(* IEC 61131-3 sources: 3D-Asset-Platform-V2/openplc/cobot-6dof-smart-demo, 5 files *)

(* ---- cobot_6dof_iot_condition_monitoring.st ---- *)
VAR
  Command AT %QW90 : UINT := 0;
  Status AT %QW91 : UINT := 0;
  ActiveStep AT %QW92 : UINT := 0;
  ElapsedMsOut AT %QW93 : UINT := 0;
  AlarmCode AT %QW94 : UINT := 0;
  ConditionState AT %QW95 : UINT := 3;
  SpeedPermille AT %QW96 : UINT := 0;
  J1Raw AT %QW100 : INT := 0;
  J2Raw AT %QW101 : INT := -6109;
  J3Raw AT %QW102 : INT := 13090;
  J4Raw AT %QW103 : INT := 8727;
  J5Raw AT %QW104 : INT := 0;
  J6Raw AT %QW105 : INT := 0;
  TemperatureCx100 AT %QW120 : INT := 0;
  HumidityRHx100 AT %QW121 : UINT := 0;
  GyroDpsx100 AT %QW122 : UINT := 0;
  SensorAgeMs AT %QW123 : UINT := 65535;
  SensorValid AT %QW124 : UINT := 0;
  SensorSequence AT %QW125 : UINT := 0;
  SensorQualityBits AT %QW126 : UINT := 0;
  SensorPolicy AT %QW127 : UINT := 1;
  CycleTimer : TON;
  MotionIdleTimer : TON;
  TimerEnabled : BOOL := FALSE;
  ResetTimer : BOOL := TRUE;
  ElapsedMs : DINT := 0;
  SegmentStartMs : DINT := 0;
  SegmentDurationMs : DINT := 1;
  P : REAL := 0.0;
  MotionScale : REAL := 1.0;
  TemperatureC : REAL := 0.0;
  HumidityRH : REAL := 0.0;
  GyroDps : REAL := 0.0;
  J1Deg : REAL := 0.0;
  J2Deg : REAL := -35.0;
  J3Deg : REAL := 75.0;
  J4Deg : REAL := 50.0;
  J5Deg : REAL := 0.0;
  J6Deg : REAL := 0.0;
  TargetJ1 : REAL := 0.0;
  TargetJ2 : REAL := -35.0;
  TargetJ3 : REAL := 75.0;
  TargetJ4 : REAL := 50.0;
  TargetJ5 : REAL := 0.0;
  TargetJ6 : REAL := 0.0;
  MotionPresent : BOOL := FALSE;
  DegToRadScaled : REAL := 174.5329;
END_VAR

TemperatureC := INT_TO_REAL(TemperatureCx100) / 100.0;
HumidityRH := UINT_TO_REAL(HumidityRHx100) / 100.0;
GyroDps := UINT_TO_REAL(GyroDpsx100) / 100.0;
MotionPresent := GyroDps >= 3.0;
MotionIdleTimer(IN := (SensorPolicy = 1) AND (NOT MotionPresent), PT := T#2s);

ConditionState := 0;
AlarmCode := 0;
MotionScale := 1.0;
SpeedPermille := 1000;

IF (SensorValid = 0) OR ((SensorQualityBits AND 1) = 0) OR (SensorAgeMs > 2500) THEN
  ConditionState := 3;
  AlarmCode := 4;
  MotionScale := 0.0;
  SpeedPermille := 0;
ELSIF (SensorPolicy = 1) AND ((SensorQualityBits AND 16) = 0) THEN
  ConditionState := 3;
  AlarmCode := 6;
  MotionScale := 0.0;
  SpeedPermille := 0;
ELSIF (SensorPolicy = 1) AND MotionIdleTimer.Q THEN
  ConditionState := 2;
  AlarmCode := 5;
  MotionScale := 0.0;
  SpeedPermille := 0;
ELSIF (TemperatureC >= 55.0) OR (HumidityRH >= 85.0) OR (GyroDps >= 220.0) THEN
  ConditionState := 2;
  MotionScale := 0.0;
  SpeedPermille := 0;
  IF TemperatureC >= 55.0 THEN
    AlarmCode := 1;
  ELSIF HumidityRH >= 85.0 THEN
    AlarmCode := 2;
  ELSE
    AlarmCode := 3;
  END_IF;
ELSIF (TemperatureC >= 45.0) OR (HumidityRH >= 75.0) OR (GyroDps >= 120.0) THEN
  ConditionState := 1;
  MotionScale := 0.55;
  SpeedPermille := 550;
END_IF;

IF Command = 2 THEN
  TimerEnabled := FALSE;
  ResetTimer := TRUE;
  Status := 2;
  ActiveStep := 0;
  ElapsedMsOut := 0;
  J1Deg := 0.0;
  J2Deg := -35.0;
  J3Deg := 75.0;
  J4Deg := 50.0;
  J5Deg := 0.0;
  J6Deg := 0.0;
ELSIF Command = 0 THEN
  TimerEnabled := FALSE;
  ResetTimer := TRUE;
  Status := 0;
  ActiveStep := 0;
  J1Deg := INT_TO_REAL(J1Raw) / DegToRadScaled;
  J2Deg := INT_TO_REAL(J2Raw) / DegToRadScaled;
  J3Deg := INT_TO_REAL(J3Raw) / DegToRadScaled;
  J4Deg := INT_TO_REAL(J4Raw) / DegToRadScaled;
  J5Deg := INT_TO_REAL(J5Raw) / DegToRadScaled;
  J6Deg := INT_TO_REAL(J6Raw) / DegToRadScaled;
ELSIF ConditionState >= 2 THEN
  TimerEnabled := FALSE;
  ResetTimer := TRUE;
  Status := 3;
  ActiveStep := 0;
ELSE
  Status := 1;
  IF ResetTimer THEN
    TimerEnabled := FALSE;
    ResetTimer := FALSE;
  ELSE
    TimerEnabled := TRUE;
  END_IF;

  CycleTimer(IN := TimerEnabled, PT := T#12s);
  ElapsedMs := TIME_TO_DINT(CycleTimer.ET);
  IF ElapsedMs > 12000 THEN ElapsedMs := 12000; END_IF;
  ElapsedMsOut := DINT_TO_UINT(ElapsedMs);

  IF ElapsedMs < 3000 THEN
    ActiveStep := 1; SegmentStartMs := 0; SegmentDurationMs := 3000;
    TargetJ1 := -90.0; TargetJ2 := -10.0; TargetJ3 := 105.0;
    TargetJ4 := 10.0; TargetJ5 := -45.0; TargetJ6 := -90.0;
  ELSIF ElapsedMs < 6000 THEN
    ActiveStep := 2; SegmentStartMs := 3000; SegmentDurationMs := 3000;
    TargetJ1 := 90.0; TargetJ2 := 40.0; TargetJ3 := 125.0;
    TargetJ4 := -70.0; TargetJ5 := 60.0; TargetJ6 := 120.0;
  ELSIF ElapsedMs < 9000 THEN
    ActiveStep := 3; SegmentStartMs := 6000; SegmentDurationMs := 3000;
    TargetJ1 := -55.0; TargetJ2 := -75.0; TargetJ3 := 45.0;
    TargetJ4 := 120.0; TargetJ5 := -80.0; TargetJ6 := -140.0;
  ELSE
    ActiveStep := 4; SegmentStartMs := 9000; SegmentDurationMs := 3000;
    TargetJ1 := 0.0; TargetJ2 := -35.0; TargetJ3 := 75.0;
    TargetJ4 := 50.0; TargetJ5 := 0.0; TargetJ6 := 0.0;
  END_IF;

  P := DINT_TO_REAL(ElapsedMs - SegmentStartMs) / DINT_TO_REAL(SegmentDurationMs);
  IF P < 0.0 THEN P := 0.0; END_IF;
  IF P > 1.0 THEN P := 1.0; END_IF;
  P := P * P * (3.0 - (2.0 * P));

  J1Deg := J1Deg + (((0.0 + ((TargetJ1 - 0.0) * MotionScale)) - J1Deg) * P);
  J2Deg := J2Deg + (((-35.0 + ((TargetJ2 - (-35.0)) * MotionScale)) - J2Deg) * P);
  J3Deg := J3Deg + (((75.0 + ((TargetJ3 - 75.0) * MotionScale)) - J3Deg) * P);
  J4Deg := J4Deg + (((50.0 + ((TargetJ4 - 50.0) * MotionScale)) - J4Deg) * P);
  J5Deg := J5Deg + (((0.0 + ((TargetJ5 - 0.0) * MotionScale)) - J5Deg) * P);
  J6Deg := J6Deg + (((0.0 + ((TargetJ6 - 0.0) * MotionScale)) - J6Deg) * P);

  IF CycleTimer.Q THEN ResetTimer := TRUE; END_IF;
END_IF;

J1Raw := REAL_TO_INT(J1Deg * DegToRadScaled);
J2Raw := REAL_TO_INT(J2Deg * DegToRadScaled);
J3Raw := REAL_TO_INT(J3Deg * DegToRadScaled);
J4Raw := REAL_TO_INT(J4Deg * DegToRadScaled);
J5Raw := REAL_TO_INT(J5Deg * DegToRadScaled);
J6Raw := REAL_TO_INT(J6Deg * DegToRadScaled);

(* ---- cobot_6dof_smart_demo.st ---- *)
VAR
  Command AT %QW90 : UINT := 1;
  Status AT %QW91 : UINT := 1;
  ActiveStep AT %QW92 : UINT := 0;
  ElapsedMsOut AT %QW93 : UINT := 0;
  J1Raw AT %QW100 : INT := 0;
  J2Raw AT %QW101 : INT := -6109;
  J3Raw AT %QW102 : INT := 13090;
  J4Raw AT %QW103 : INT := 8727;
  J5Raw AT %QW104 : INT := 0;
  J6Raw AT %QW105 : INT := 0;
  CycleTimer : TON;
  TimerEnabled : BOOL := TRUE;
  ResetTimer : BOOL := FALSE;
  ElapsedMs : DINT := 0;
  SegmentStartMs : DINT := 0;
  SegmentDurationMs : DINT := 1;
  P : REAL := 0.0;
  J1Deg : REAL := 0.0;
  J2Deg : REAL := -35.0;
  J3Deg : REAL := 75.0;
  J4Deg : REAL := 50.0;
  J5Deg : REAL := 0.0;
  J6Deg : REAL := 0.0;
  DegToRadScaled : REAL := 174.5329;
END_VAR

IF Command = 2 THEN
  TimerEnabled := FALSE; Status := 2; ActiveStep := 0; ElapsedMsOut := 0;
  J1Deg := 0.0; J2Deg := -35.0; J3Deg := 75.0;
  J4Deg := 50.0; J5Deg := 0.0; J6Deg := 0.0;
ELSIF Command = 0 THEN
  TimerEnabled := FALSE; Status := 0; ActiveStep := 0;
  J1Deg := INT_TO_REAL(J1Raw) / DegToRadScaled;
  J2Deg := INT_TO_REAL(J2Raw) / DegToRadScaled;
  J3Deg := INT_TO_REAL(J3Raw) / DegToRadScaled;
  J4Deg := INT_TO_REAL(J4Raw) / DegToRadScaled;
  J5Deg := INT_TO_REAL(J5Raw) / DegToRadScaled;
  J6Deg := INT_TO_REAL(J6Raw) / DegToRadScaled;
ELSE
  Status := 1;
  IF ResetTimer THEN
    TimerEnabled := FALSE; ResetTimer := FALSE;
  ELSE
    TimerEnabled := TRUE;
  END_IF;

  CycleTimer(IN := TimerEnabled, PT := T#10s);
  ElapsedMs := TIME_TO_DINT(CycleTimer.ET);
  IF ElapsedMs > 10000 THEN ElapsedMs := 10000; END_IF;
  ElapsedMsOut := DINT_TO_UINT(ElapsedMs);

  IF ElapsedMs < 1400 THEN
    ActiveStep := 1; SegmentStartMs := 0; SegmentDurationMs := 1400;
  ELSIF ElapsedMs < 2400 THEN
    ActiveStep := 2; SegmentStartMs := 1400; SegmentDurationMs := 1000;
  ELSIF ElapsedMs < 3200 THEN
    ActiveStep := 3; SegmentStartMs := 2400; SegmentDurationMs := 800;
  ELSIF ElapsedMs < 5600 THEN
    ActiveStep := 4; SegmentStartMs := 3200; SegmentDurationMs := 2400;
  ELSIF ElapsedMs < 7600 THEN
    ActiveStep := 5; SegmentStartMs := 5600; SegmentDurationMs := 2000;
  ELSE
    ActiveStep := 6; SegmentStartMs := 7600; SegmentDurationMs := 2400;
  END_IF;

  IF SegmentDurationMs > 0 THEN
    P := DINT_TO_REAL(ElapsedMs - SegmentStartMs) / DINT_TO_REAL(SegmentDurationMs);
    IF P < 0.0 THEN P := 0.0; ELSIF P > 1.0 THEN P := 1.0; END_IF;
    P := P * P * (3.0 - (2.0 * P));
  ELSE
    P := 0.0;
  END_IF;

  IF ActiveStep = 1 THEN
    J1Deg := 0.0 + ((-55.0 - 0.0) * P);
    J2Deg := -35.0 + ((-10.0 - (-35.0)) * P);
    J3Deg := 75.0 + ((85.0 - 75.0) * P);
    J4Deg := 50.0 + ((25.0 - 50.0) * P);
    J5Deg := 0.0;
    J6Deg := 0.0;
  ELSIF ActiveStep = 2 THEN
    J1Deg := -55.0;
    J2Deg := -10.0 + ((15.0 - (-10.0)) * P);
    J3Deg := 85.0 + ((80.0 - 85.0) * P);
    J4Deg := 25.0 + ((-5.0 - 25.0) * P);
    J5Deg := 0.0;
    J6Deg := 0.0;
  ELSIF ActiveStep = 3 THEN
    J1Deg := -55.0;
    J2Deg := 15.0;
    J3Deg := 80.0;
    J4Deg := -5.0;
    J5Deg := 0.0;
    J6Deg := 0.0 + ((90.0 - 0.0) * P);
  ELSIF ActiveStep = 4 THEN
    J1Deg := -55.0 + ((50.0 - (-55.0)) * P);
    J2Deg := 15.0 + ((-10.0 - 15.0) * P);
    J3Deg := 80.0 + ((85.0 - 80.0) * P);
    J4Deg := -5.0 + ((25.0 - (-5.0)) * P);
    J5Deg := 0.0;
    J6Deg := 90.0;
  ELSIF ActiveStep = 5 THEN
    J1Deg := 50.0;
    J2Deg := -10.0 + ((15.0 - (-10.0)) * P);
    J3Deg := 85.0 + ((80.0 - 85.0) * P);
    J4Deg := 25.0 + ((-5.0 - 25.0) * P);
    J5Deg := 0.0 + ((30.0 - 0.0) * P);
    J6Deg := 90.0 + ((-90.0 - 90.0) * P);
  ELSE
    J1Deg := 50.0 + ((0.0 - 50.0) * P);
    J2Deg := 15.0 + ((-35.0 - 15.0) * P);
    J3Deg := 80.0 + ((75.0 - 80.0) * P);
    J4Deg := -5.0 + ((50.0 - (-5.0)) * P);
    J5Deg := 30.0 + ((0.0 - 30.0) * P);
    J6Deg := -90.0 + ((0.0 - (-90.0)) * P);
  END_IF;

  IF CycleTimer.Q THEN ResetTimer := TRUE; END_IF;
END_IF;

J1Raw := REAL_TO_INT(J1Deg * DegToRadScaled);
J2Raw := REAL_TO_INT(J2Deg * DegToRadScaled);
J3Raw := REAL_TO_INT(J3Deg * DegToRadScaled);
J4Raw := REAL_TO_INT(J4Deg * DegToRadScaled);
J5Raw := REAL_TO_INT(J5Deg * DegToRadScaled);
J6Raw := REAL_TO_INT(J6Deg * DegToRadScaled);

(* ---- cobot_6dof_smart_demo_amplified.st ---- *)
VAR
  Command AT %QW90 : UINT := 0;
  Status AT %QW91 : UINT := 0;
  ActiveStep AT %QW92 : UINT := 0;
  ElapsedMsOut AT %QW93 : UINT := 0;
  J1Raw AT %QW100 : INT := 0;
  J2Raw AT %QW101 : INT := -6109;
  J3Raw AT %QW102 : INT := 13090;
  J4Raw AT %QW103 : INT := 8727;
  J5Raw AT %QW104 : INT := 0;
  J6Raw AT %QW105 : INT := 0;
  CycleTimer : TON;
  TimerEnabled : BOOL := FALSE;
  ResetTimer : BOOL := FALSE;
  ElapsedMs : DINT := 0;
  SegmentStartMs : DINT := 0;
  SegmentDurationMs : DINT := 1;
  P : REAL := 0.0;
  J1Deg : REAL := 0.0;
  J2Deg : REAL := -35.0;
  J3Deg : REAL := 75.0;
  J4Deg : REAL := 50.0;
  J5Deg : REAL := 0.0;
  J6Deg : REAL := 0.0;
  DegToRadScaled : REAL := 174.5329;
END_VAR

IF Command = 2 THEN
  TimerEnabled := FALSE;
  ResetTimer := TRUE;
  Status := 2;
  ActiveStep := 0;
  ElapsedMsOut := 0;
  J1Deg := 0.0;
  J2Deg := -35.0;
  J3Deg := 75.0;
  J4Deg := 50.0;
  J5Deg := 0.0;
  J6Deg := 0.0;
ELSIF Command = 0 THEN
  TimerEnabled := FALSE;
  ResetTimer := TRUE;
  Status := 0;
  ActiveStep := 0;
  ElapsedMsOut := 0;
  J1Deg := INT_TO_REAL(J1Raw) / DegToRadScaled;
  J2Deg := INT_TO_REAL(J2Raw) / DegToRadScaled;
  J3Deg := INT_TO_REAL(J3Raw) / DegToRadScaled;
  J4Deg := INT_TO_REAL(J4Raw) / DegToRadScaled;
  J5Deg := INT_TO_REAL(J5Raw) / DegToRadScaled;
  J6Deg := INT_TO_REAL(J6Raw) / DegToRadScaled;
ELSE
  Status := 1;

  IF ResetTimer THEN
    TimerEnabled := FALSE;
    ResetTimer := FALSE;
  ELSE
    TimerEnabled := TRUE;
  END_IF;

  CycleTimer(IN := TimerEnabled, PT := T#18s);
  ElapsedMs := TIME_TO_DINT(CycleTimer.ET);
  IF ElapsedMs > 18000 THEN ElapsedMs := 18000; END_IF;
  ElapsedMsOut := DINT_TO_UINT(ElapsedMs);

  IF ElapsedMs < 3000 THEN
    ActiveStep := 1;
    SegmentStartMs := 0;
    SegmentDurationMs := 3000;
  ELSIF ElapsedMs < 6000 THEN
    ActiveStep := 2;
    SegmentStartMs := 3000;
    SegmentDurationMs := 3000;
  ELSIF ElapsedMs < 9000 THEN
    ActiveStep := 3;
    SegmentStartMs := 6000;
    SegmentDurationMs := 3000;
  ELSIF ElapsedMs < 12000 THEN
    ActiveStep := 4;
    SegmentStartMs := 9000;
    SegmentDurationMs := 3000;
  ELSIF ElapsedMs < 15000 THEN
    ActiveStep := 5;
    SegmentStartMs := 12000;
    SegmentDurationMs := 3000;
  ELSE
    ActiveStep := 6;
    SegmentStartMs := 15000;
    SegmentDurationMs := 3000;
  END_IF;

  P := DINT_TO_REAL(ElapsedMs - SegmentStartMs) / DINT_TO_REAL(SegmentDurationMs);
  IF P < 0.0 THEN P := 0.0; END_IF;
  IF P > 1.0 THEN P := 1.0; END_IF;
  P := P * P * (3.0 - (2.0 * P));

  IF ActiveStep = 1 THEN
    J1Deg := 0.0 + ((-150.0 - 0.0) * P);
    J2Deg := -35.0 + ((-75.0 - (-35.0)) * P);
    J3Deg := 75.0 + ((110.0 - 75.0) * P);
    J4Deg := 50.0 + ((-90.0 - 50.0) * P);
    J5Deg := 0.0 + ((-80.0 - 0.0) * P);
    J6Deg := 0.0 + ((-160.0 - 0.0) * P);
  ELSIF ActiveStep = 2 THEN
    J1Deg := -150.0;
    J2Deg := -75.0 + ((70.0 - (-75.0)) * P);
    J3Deg := 110.0 + ((145.0 - 110.0) * P);
    J4Deg := -90.0 + ((120.0 - (-90.0)) * P);
    J5Deg := -80.0 + ((100.0 - (-80.0)) * P);
    J6Deg := -160.0 + ((160.0 - (-160.0)) * P);
  ELSIF ActiveStep = 3 THEN
    J1Deg := -150.0 + ((150.0 - (-150.0)) * P);
    J2Deg := 70.0 + ((20.0 - 70.0) * P);
    J3Deg := 145.0 + ((40.0 - 145.0) * P);
    J4Deg := 120.0 + ((-130.0 - 120.0) * P);
    J5Deg := 100.0 + ((-110.0 - 100.0) * P);
    J6Deg := 160.0 + ((-170.0 - 160.0) * P);
  ELSIF ActiveStep = 4 THEN
    J1Deg := 150.0;
    J2Deg := 20.0 + ((-100.0 - 20.0) * P);
    J3Deg := 40.0 + ((130.0 - 40.0) * P);
    J4Deg := -130.0 + ((140.0 - (-130.0)) * P);
    J5Deg := -110.0 + ((120.0 - (-110.0)) * P);
    J6Deg := -170.0 + ((170.0 - (-170.0)) * P);
  ELSIF ActiveStep = 5 THEN
    J1Deg := 150.0 + ((-110.0 - 150.0) * P);
    J2Deg := -100.0 + ((80.0 - (-100.0)) * P);
    J3Deg := 130.0 + ((25.0 - 130.0) * P);
    J4Deg := 140.0 + ((-140.0 - 140.0) * P);
    J5Deg := 120.0 + ((-120.0 - 120.0) * P);
    J6Deg := 170.0 + ((-165.0 - 170.0) * P);
  ELSE
    J1Deg := -110.0 + ((0.0 - (-110.0)) * P);
    J2Deg := 80.0 + ((-35.0 - 80.0) * P);
    J3Deg := 25.0 + ((75.0 - 25.0) * P);
    J4Deg := -140.0 + ((50.0 - (-140.0)) * P);
    J5Deg := -120.0 + ((0.0 - (-120.0)) * P);
    J6Deg := -165.0 + ((0.0 - (-165.0)) * P);
  END_IF;

  IF CycleTimer.Q THEN ResetTimer := TRUE; END_IF;
END_IF;

IF J1Deg < -170.0 THEN J1Deg := -170.0; END_IF;
IF J1Deg > 170.0 THEN J1Deg := 170.0; END_IF;
IF J2Deg < -120.0 THEN J2Deg := -120.0; END_IF;
IF J2Deg > 120.0 THEN J2Deg := 120.0; END_IF;
IF J3Deg < -170.0 THEN J3Deg := -170.0; END_IF;
IF J3Deg > 170.0 THEN J3Deg := 170.0; END_IF;
IF J4Deg < -170.0 THEN J4Deg := -170.0; END_IF;
IF J4Deg > 170.0 THEN J4Deg := 170.0; END_IF;
IF J5Deg < -170.0 THEN J5Deg := -170.0; END_IF;
IF J5Deg > 170.0 THEN J5Deg := 170.0; END_IF;
IF J6Deg < -175.0 THEN J6Deg := -175.0; END_IF;
IF J6Deg > 175.0 THEN J6Deg := 175.0; END_IF;

J1Raw := REAL_TO_INT(J1Deg * DegToRadScaled);
J2Raw := REAL_TO_INT(J2Deg * DegToRadScaled);
J3Raw := REAL_TO_INT(J3Deg * DegToRadScaled);
J4Raw := REAL_TO_INT(J4Deg * DegToRadScaled);
J5Raw := REAL_TO_INT(J5Deg * DegToRadScaled);
J6Raw := REAL_TO_INT(J6Deg * DegToRadScaled);

(* ---- cobot_6dof_smart_demo_rectificado.st ---- *)
VAR
  Command AT %QW90 : UINT := 1;
  Status AT %QW91 : UINT := 1;
  ActiveStep AT %QW92 : UINT := 0;
  ElapsedMsOut AT %QW93 : UINT := 0;
  J1Raw AT %QW100 : INT := 0;
  J2Raw AT %QW101 : INT := -6109;
  J3Raw AT %QW102 : INT := 13090;
  J4Raw AT %QW103 : INT := 8727;
  J5Raw AT %QW104 : INT := 0;
  J6Raw AT %QW105 : INT := 0;
  CycleTimer : TON;
  TimerEnabled : BOOL := TRUE;
  ResetTimer : BOOL := FALSE;
  ElapsedMs : DINT := 0;
  SegmentStartMs : DINT := 0;
  SegmentDurationMs : DINT := 1;
  P : REAL := 0.0;
  J1Deg : REAL := 0.0;
  J2Deg : REAL := -35.0;
  J3Deg : REAL := 75.0;
  J4Deg : REAL := 50.0;
  J5Deg : REAL := 0.0;
  J6Deg : REAL := 0.0;
  DegToRadScaled : REAL := 174.5329;
END_VAR

IF Command = 2 THEN
  TimerEnabled := FALSE; Status := 2; ActiveStep := 0; ElapsedMsOut := 0;
  J1Deg := 0.0; J2Deg := -35.0; J3Deg := 75.0;
  J4Deg := 50.0; J5Deg := 0.0; J6Deg := 0.0;
ELSIF Command = 0 THEN
  TimerEnabled := FALSE; Status := 0; ActiveStep := 0;
  J1Deg := INT_TO_REAL(J1Raw) / DegToRadScaled;
  J2Deg := INT_TO_REAL(J2Raw) / DegToRadScaled;
  J3Deg := INT_TO_REAL(J3Raw) / DegToRadScaled;
  J4Deg := INT_TO_REAL(J4Raw) / DegToRadScaled;
  J5Deg := INT_TO_REAL(J5Raw) / DegToRadScaled;
  J6Deg := INT_TO_REAL(J6Raw) / DegToRadScaled;
ELSE
  Status := 1;
  IF ResetTimer THEN
    TimerEnabled := FALSE; ResetTimer := FALSE;
  ELSE
    TimerEnabled := TRUE;
  END_IF;

  CycleTimer(IN := TimerEnabled, PT := T#10s);
  ElapsedMs := TIME_TO_DINT(CycleTimer.ET);
  IF ElapsedMs > 10000 THEN ElapsedMs := 10000; END_IF;
  ElapsedMsOut := DINT_TO_UINT(ElapsedMs);

  IF ElapsedMs < 1400 THEN
    ActiveStep := 1; SegmentStartMs := 0; SegmentDurationMs := 1400;
  ELSIF ElapsedMs < 2400 THEN
    ActiveStep := 2; SegmentStartMs := 1400; SegmentDurationMs := 1000;
  ELSIF ElapsedMs < 3200 THEN
    ActiveStep := 3; SegmentStartMs := 2400; SegmentDurationMs := 800;
  ELSIF ElapsedMs < 5600 THEN
    ActiveStep := 4; SegmentStartMs := 3200; SegmentDurationMs := 2400;
  ELSIF ElapsedMs < 7600 THEN
    ActiveStep := 5; SegmentStartMs := 5600; SegmentDurationMs := 2000;
  ELSE
    ActiveStep := 6; SegmentStartMs := 7600; SegmentDurationMs := 2400;
  END_IF;

  IF SegmentDurationMs > 0 THEN
    P := DINT_TO_REAL(ElapsedMs - SegmentStartMs) / DINT_TO_REAL(SegmentDurationMs);
    IF P < 0.0 THEN P := 0.0; ELSIF P > 1.0 THEN P := 1.0; END_IF;
  ELSE
    P := 0.0;
  END_IF;

  IF ActiveStep = 1 THEN
    J1Deg := 0.0 + ((-55.0 - 0.0) * P);
    J2Deg := -35.0 + ((-10.0 - (-35.0)) * P);
    J3Deg := 75.0 + ((85.0 - 75.0) * P);
    J4Deg := 50.0 + ((25.0 - 50.0) * P);
    J5Deg := 0.0;
    J6Deg := 0.0;
  ELSIF ActiveStep = 2 THEN
    J1Deg := -55.0;
    J2Deg := -10.0 + ((15.0 - (-10.0)) * P);
    J3Deg := 85.0 + ((80.0 - 85.0) * P);
    J4Deg := 25.0 + ((-5.0 - 25.0) * P);
    J5Deg := 0.0;
    J6Deg := 0.0;
  ELSIF ActiveStep = 3 THEN
    J1Deg := -55.0;
    J2Deg := 15.0;
    J3Deg := 80.0;
    J4Deg := -5.0;
    J5Deg := 0.0;
    J6Deg := 0.0 + ((90.0 - 0.0) * P);
  ELSIF ActiveStep = 4 THEN
    J1Deg := -55.0 + ((50.0 - (-55.0)) * P);
    J2Deg := 15.0 + ((-10.0 - 15.0) * P);
    J3Deg := 80.0 + ((85.0 - 80.0) * P);
    J4Deg := -5.0 + ((25.0 - (-5.0)) * P);
    J5Deg := 0.0;
    J6Deg := 90.0;
  ELSIF ActiveStep = 5 THEN
    J1Deg := 50.0;
    J2Deg := -10.0 + ((15.0 - (-10.0)) * P);
    J3Deg := 85.0 + ((80.0 - 85.0) * P);
    J4Deg := 25.0 + ((-5.0 - 25.0) * P);
    J5Deg := 0.0 + ((30.0 - 0.0) * P);
    J6Deg := 90.0 + ((-90.0 - 90.0) * P);
  ELSE
    J1Deg := 50.0 + ((0.0 - 50.0) * P);
    J2Deg := 15.0 + ((-35.0 - 15.0) * P);
    J3Deg := 80.0 + ((75.0 - 80.0) * P);
    J4Deg := -5.0 + ((50.0 - (-5.0)) * P);
    J5Deg := 30.0 + ((0.0 - 30.0) * P);
    J6Deg := -90.0 + ((0.0 - (-90.0)) * P);
  END_IF;

  IF CycleTimer.Q THEN ResetTimer := TRUE; END_IF;
END_IF;

J1Raw := REAL_TO_INT(J1Deg * DegToRadScaled);
J2Raw := REAL_TO_INT(J2Deg * DegToRadScaled);
J3Raw := REAL_TO_INT(J3Deg * DegToRadScaled);
J4Raw := REAL_TO_INT(J4Deg * DegToRadScaled);
J5Raw := REAL_TO_INT(J5Deg * DegToRadScaled);
J6Raw := REAL_TO_INT(J6Deg * DegToRadScaled);

(* ---- watertank.st ---- *)
  VAR
    openOutletValve : BOOL AT %QX0.1;
    openInletValve : BOOL AT %QX0.4;
    outletValveOpenStatus : BOOL AT %QX0.3;
    inletValveOpenStatus : BOOL AT %QX0.5;
    airValveOpenStatus : BOOL AT %QX0.6;
    level : INT AT %IW2;
    level_max : INT AT %IW3;
    level_min : INT := 10;
  END_VAR

IF (level >= level_max) AND airValveOpenStatus THEN
  openOutletValve := TRUE;
  outletValveOpenStatus := TRUE;
  openInletValve := FALSE;
  inletValveOpenStatus := FALSE;
END_IF;

IF (level < (level_max - level_min)) AND airValveOpenStatus THEN
  openOutletValve := FALSE;
  outletValveOpenStatus := FALSE;
  openInletValve := TRUE;
  inletValveOpenStatus := TRUE;
END_IF;

IF NOT airValveOpenStatus THEN
  openOutletValve := FALSE;
  outletValveOpenStatus := FALSE;
  openInletValve := FALSE;
  inletValveOpenStatus := FALSE;
END_IF;
